PROGRAM MAIN
VAR
END_VAR

ACTION motor:

END_ACTION

END_PROGRAM

(* stored: Version 1.1.0.1, ProductVersion 3.1.4024.9
   POU MAIN: Id {082901b3-abcc-478c-8f65-6930cc000521}, SpecialFunc None
   Action motor: Id {cdd9b3f3-26f6-4587-9151-2f12ff38b31e} *)
